FUNCTION FC_WithAction : DINT
VAR_INPUT
    nInput : DINT;
    bProcess : BOOL;
END_VAR
VAR
    nResult : DINT;
END_VAR

nResult := nInput;

IF bProcess THEN
    nResult := nResult * 2;
END_IF;

FC_WithAction := nResult;

ACTION ProcessArray:
nLocalSum := 0;

FOR i := 0 TO 9 DO
    IF i MOD 2 = 0 THEN
        nLocalSum := nLocalSum + i;
    END_IF;
END_FOR;

WHILE nLocalSum > 100 DO
    nLocalSum := nLocalSum - 10;
END_WHILE;

nResult := nLocalSum;
END_ACTION

END_FUNCTION

(* stored: Version 1.1.0.1
   POU FC_WithAction: Id {55555555-5555-5555-5555-555555555555}, SpecialFunc None
   Action ProcessArray: Id {aaaaaaaa-1111-2222-3333-444444444444} *)
